INTERFACE I_Object EXTENDS __SYSTEM.IQueryInterface

METHOD Equals : BOOL
VAR_INPUT
    ipObject:       I_Object;
END_VAR
END_METHOD

PROPERTY nIdentity : ULINT
GET
END_GET
END_PROPERTY

PROPERTY sPath : STRING(MAX_STRING_LENGTH)
GET
END_GET
END_PROPERTY

END_INTERFACE

(* stored: Version 1.1.0.1, ProductVersion 3.1.4024.12
   Itf I_Object: Id {96c915d9-541c-4566-8f01-7492919705b5}
   Method Equals: Id {268e9796-2d0c-0dbe-24e3-c35c5e029c1c}
   Property nIdentity: Id {92b56106-a7b5-4964-b45c-98b59de921b1}
   Get Get: Id {0bd6f9ae-19ae-44ce-9d71-fb8d6bfead8a}
   Property sPath: Id {703fc0af-c533-4d23-89ec-6b8f676dca77}
   Get Get: Id {4521e10c-7e6c-46c5-81a0-1856018e854b} *)
